FUNCTION_BLOCK FB_TestRound EXTENDS TcUnit.FB_TestSuite

//REAL
testRoundRealFail();
testRoundRealSuccess();
testRoundRealToHigh();
testRoundRealToHigh2();

// LREAL
testRoundLREALFail();
testRoundLREALSuccess();
testRoundLREALToHigh();
testRoundLREALToHigh2();

// Negative LREAL
testRoundLREALNegative();
testRoundLREALNegativeToHigh();

// Negative REAL
testRoundREALNegative();
testRoundREALNegativeToHigh();

METHOD testRoundLREALFail
VAR
	rValue 		: LREAL := 1000.222222;
	Actual		: LREAL;
	Expected  	: LREAL;
END_VAR
TEST('testRoundLREALFail');

// Act
Actual := 1000.222; 

// Arrange
Expected := 1000.22;

// Assert
AssertFalse( Condition := Expected = Actual, 
			 Message := 'testRoundLREALFail Failed to round LREAL');
			 
			 
			 
TEST_FINISHED();
END_METHOD

METHOD testRoundLREALNegative
VAR
	rValue 		: LREAL := -1000.22;
	Actual		: LREAL;
	Expected  	: LREAL;
END_VAR
TEST('testRoundLREALNegative');

// Act
Actual := F_ROUND_LREAL(rValue, 1); 

// Arrange
Expected := -1000.2;

// Assert
AssertEquals_LREAL( Expected :=  Expected, 
				Actual := Actual,
				Delta := 0.00,
			 	Message := 'testRoundLREALNegative Failed to round LREAL Negative');
			 
			 
			 
TEST_FINISHED();
END_METHOD

METHOD testRoundLREALNegativeToHigh
VAR
	rValue 		: LREAL := -1000.556;
	Actual		: LREAL;
	Expected  	: LREAL;
END_VAR
TEST('testRoundLREALNegativeToHigh');

// Act
Actual := F_ROUND_LREAL(rValue, 2); 

// Arrange
Expected := -1000.56;

// Assert
AssertEquals_LREAL( Expected :=  Expected, 
				Actual := Actual,
				Delta := 0.00,
			 	Message := 'testRoundLREALNegativeToHigh Failed to round LREAL Negative');
			 
			 
			 
TEST_FINISHED();
END_METHOD

METHOD testRoundLREALSuccess
VAR
	rValue 		: LREAL := 1000.222222;
	Actual		: LREAL;
	Expected  	: LREAL;
END_VAR
TEST('testRoundLREALSuccess');

// Act
Actual := F_ROUND_LREAL(rValue, 2); 

// Arrange
Expected := 1000.22;

// Assert
AssertEquals(Expected := Expected, 
			 Actual := Actual,
			 Message := 'testRoundLREALSuccess Failed to round LREAL');
			 
			 
			 
TEST_FINISHED();
END_METHOD

METHOD testRoundLREALToHigh
VAR
	rValue 		: LREAL := 1000.226666;
	Actual		: LREAL;
	Expected  	: LREAL;
END_VAR
TEST('testRoundLREALToHigh');

// Act
Actual := F_ROUND_LREAL(rValue, 2); 

// Arrange
Expected := 1000.23;

// Assert
AssertEquals_LREAL( Expected :=  Expected, 
				Actual := Actual,
				Delta := 0.00,
			 	Message := 'testRoundLREALToHigh Failed to round LREAL');
			 
			 
			 
TEST_FINISHED();
END_METHOD

METHOD testRoundLREALToHigh2
VAR
	rValue 		: LREAL := 1000.95;
	Actual		: LREAL;
	Expected  	: LREAL;
END_VAR
TEST('testRoundLREALToHigh2');

// Act
Actual := F_ROUND_LREAL(rValue, 1); 

// Arrange
Expected := 1001.0;

// Assert
AssertEquals_LREAL( Expected :=  Expected, 
				Actual := Actual,
				Delta := 0.00,
			 	Message := 'testRoundLREALToHigh2 Failed to round LREAL');
			 
			 
			 
TEST_FINISHED();
END_METHOD

METHOD testRoundRealFail
VAR
	rValue 		: REAL := 1000.222222;
	Actual		: REAL;
	Expected  	: REAL;
END_VAR
TEST('testRoundRealFail');

// Act
Actual := 1000.222; 

// Arrange
Expected := 1000.22;

// Assert
AssertFalse( Condition := Expected = Actual, 
			 Message := 'testRoundRealFail Failed to round REAL');
			 
			 
			 
TEST_FINISHED();
END_METHOD

METHOD testRoundRealNegative
VAR
	rValue 		: REAL := -1000.22;
	Actual		: REAL;
	Expected  	: REAL;
END_VAR
TEST('testRoundRealNegative');

// Act
Actual := F_ROUND_REAL(rValue, 1); 

// Arrange
Expected := -1000.2;

// Assert
AssertEquals_REAL( Expected :=  Expected, 
				Actual := Actual,
				Delta := 0.00,
			 	Message := 'testRoundRealNegative Failed to round REAL Negative');
			 
			 
			 
TEST_FINISHED();
END_METHOD

METHOD testRoundRealNegativeToHigh
VAR
	rValue 		: REAL := -1000.556;
	Actual		: REAL;
	Expected  	: REAL;
END_VAR
TEST('testRoundRealNegativeToHigh');

// Act
Actual := F_ROUND_REAL(rValue, 2); 

// Arrange
Expected := -1000.56;

// Assert
AssertEquals_REAL( Expected :=  Expected, 
				Actual := Actual,
				Delta := 0.00,
			 	Message := 'testRoundRealNegativeToHigh Failed to round REAL Negative');
			 
			 
			 
TEST_FINISHED();
END_METHOD

METHOD testRoundRealSuccess
VAR
	rValue 		: REAL := 1000.22222;
	Actual		: REAL;
	Expected  	: REAL;
END_VAR
TEST('testRoundRealSuccess');

// Act
Actual := F_ROUND_REAL(rValue, 2); 

// Arrange
Expected := 1000.22;

// Assert
AssertEquals(Expected := Expected, 
			 Actual := Actual,
			 Message := 'testRoundRealSuccess Failed to round REAL');
			 
			 
			 
TEST_FINISHED();
END_METHOD

METHOD testRoundRealToHigh
VAR
	rValue 		: REAL := 1000.226666;
	Actual		: REAL;
	Expected  	: REAL;
END_VAR
TEST('testRoundRealToHigh');

// Act
Actual := F_ROUND_REAL(rValue, 2); 

// Arrange
Expected := 1000.23;

// Assert
AssertEquals_REAL( Expected :=  Expected, 
				Actual := Actual,
				Delta := 0.00,
			 	Message := 'testRoundRealToHigh Failed to round REAL');
			 
			 
			 
TEST_FINISHED();
END_METHOD

METHOD testRoundRealToHigh2
VAR
	rValue 		: REAL := 1000.95;
	Actual		: REAL;
	Expected  	: REAL;
END_VAR
TEST('testRoundRealToHigh2');

// Act
Actual := F_ROUND_REAL(rValue, 1); 

// Arrange
Expected := 1001.0;

// Assert
AssertEquals_REAL( Expected :=  Expected, 
				Actual := Actual,
				Delta := 0.00,
			 	Message := 'testRoundRealToHigh2 Failed to round REAL');
			 
			 
			 
TEST_FINISHED();
END_METHOD

END_FUNCTION_BLOCK

(* stored: Version 1.1.0.1, ProductVersion 3.1.4024.9
   POU FB_TestRound: Id {d168d027-9d5e-46ed-9155-14182fbf4f27}, SpecialFunc None
   Method testRoundLREALFail: Id {0190ed15-4c58-455b-af97-ebeb1778d87e}
   Method testRoundLREALNegative: Id {c521f4a9-4a25-4344-8227-e3dba5c3586a}
   Method testRoundLREALNegativeToHigh: Id {ffdda655-afb3-4693-823b-af5ceaf7328c}
   Method testRoundLREALSuccess: Id {db3ba594-9ac6-4320-9154-cadf6b53cb1a}
   Method testRoundLREALToHigh: Id {2a44110a-28bc-4805-9a4e-e040b015d8a3}
   Method testRoundLREALToHigh2: Id {77181605-9ff0-4b2c-a468-c7ebca74ce8d}
   Method testRoundRealFail: Id {6c893c88-a242-439a-98ee-31082f13b45e}
   Method testRoundRealNegative: Id {2b80e827-f24e-4139-977f-23938de9fd56}
   Method testRoundRealNegativeToHigh: Id {f2a2fc5e-a49d-48f9-a8a4-48f4ba5586ee}
   Method testRoundRealSuccess: Id {348be370-bcb0-42a0-96a8-49bab6374bd8}
   Method testRoundRealToHigh: Id {d840b773-6dc8-4f18-baa5-2e617da52be4}
   Method testRoundRealToHigh2: Id {4257ebb0-fd6a-4a94-86b6-099df61f20c3} *)
